FUNCTION_BLOCK RecipeRunner
VAR
	SetPoint : ARRAY[0..9] OF ITF_RecipePoint;
	NumberOfPoints : INT;
	BasePoint : RecipePoint := (XPoint := 0.0, YPoint := 0.0, ZPoint := 0.0);
END_VAR

METHOD AddRecipe : BOOL
VAR_INPUT
END_VAR
END_METHOD

METHOD Cycle : BOOL
VAR_INPUT
END_VAR
FOR i := 0 TO NumberOfPoints DO
	IF SetPoint[i] <> 0 THEN
		
	END_IF
END_FOR
END_METHOD

END_FUNCTION_BLOCK

(* stored: Version 1.1.0.1, ProductVersion 3.1.4024.12
   POU RecipeRunner: Id {e8e61dd5-2fc0-44f5-8efe-5a5b5f550f9b}, SpecialFunc None
   Method AddRecipe: Id {9ca0c855-cbb9-4dbd-bc81-bb9a9178075c}
   Method Cycle: Id {8390455a-4f90-48fa-b6f6-f2311414a969} *)
